(* LS Electric XG5000 project: 실습5_3로스위치 *)
(* PLC LSPLC *)

PROGRAM NewProgram (* task: 스캔 프로그램 *)
VAR
    램프1 AT %QX0.1.0 : BOOL;
    스위치1 AT %IX0.0.0 : BOOL;
    스위치2 AT %IX0.0.1 : BOOL;
END_VAR

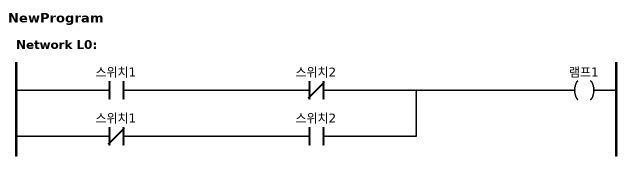
(* Rung L0 *)
램프1 := (스위치1 AND NOT 스위치2) OR (NOT 스위치1 AND 스위치2);
END_PROGRAM